FUNCTION_BLOCK PUBLIC RollerDoor
VAR_INPUT
	EN   : BOOL;
	iDoorUP    		:  BOOL;    // Clockwise Move Command 
	iDoorDOWN   	:  BOOL;    // Counterclockwise Move Command 
	iUPPosSensor  	:  BOOL;    // Forward Position sensor 180* feedback
	iDownPosSensor  :  BOOL;    // Forward Position sensor 0* feedback
END_VAR
VAR_OUTPUT
	Eno  : BOOL;
	qDoorUP		 	:  BOOL ; 	// Motor Run Status
	qDoorDown	  	:  BOOL ;    // Motor Direction Status 
END_VAR
VAR
END_VAR

// Door Safety
IF  iDoorUP AND iDoorDOWN THEN
	qDoorUP 	:= FALSE;
	qDoorDown 	:= FALSE;
END_IF

//DOOR operation
	IF iDoorUP AND NOT iUPPosSensor THEN
		qDoorUP := TRUE;
	ELSIF iDoorDOWN AND NOT iDownPosSensor THEN
		qDoorDown := TRUE;
	ELSE 
		qDoorUP := FALSE;
		qDoorDOWN := FALSE;
	END_IF

END_FUNCTION_BLOCK

(* stored: Version 1.1.0.1, ProductVersion 3.1.4024.16
   POU RollerDoor: Id {1ed1661f-21eb-4959-a6e2-faf2ecc3555f}, SpecialFunc None *)
